Fanuc KAREL source: test_form.kl

PROGRAM test_form
%NOLOCKGROUP

--lam object
%class frmpad('pathform.klc','pathform.klh','defaultpathfrm.klt')

BEGIN
END test_form
